(* LS Electric XG5000 project: 11_01_project *)
(* PLC LSPLC *)

PROGRAM NewProgram (* task: 스캔 프로그램 *)
VAR
    dd : BOOL;
    ET : TIME;
    INST : TON;
    INST1 : TP;
    INST10 : TON;
    INST11 : TMR_FLK;
    INST12 : TON;
    INST13 : TMR_FLK;
    INST14 : TOF;
    INST15 : TOF;
    INST16 : TOF;
    INST17 : TOF;
    INST18 : CTD_INT;
    INST19 : CTD_INT;
    INST2 : TP;
    INST20 : TMR_FLK;
    INST21 : TMR_FLK;
    INST22 : TOF;
    INST23 : CTD_INT;
    INST3 : TON;
    INST4 : TP;
    INST5 : TP_RST;
    INST6 : TP;
    INST7 : TMR_FLK;
    INST8 : TP;
    INST9 : TMR_FLK;
    intcv : BOOL;
    LD : BOOL;
    RST : BOOL;
    ㄱㄱ : BOOL;
    걍 : BOOL;
END_VAR

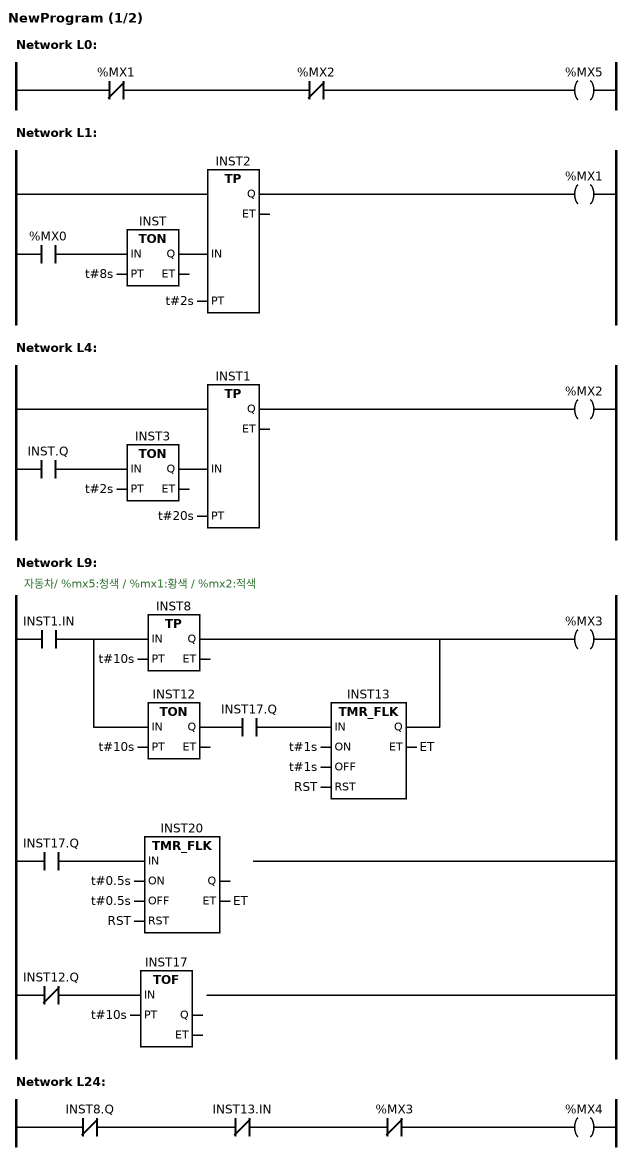
(* Rung L0 *)
%MX5 := NOT %MX1 AND NOT %MX2;
(* Rung L1 *)
INST(IN := %MX0, PT := t#8s);
INST2(IN := INST.Q, PT := t#2s);
%MX1 := INST2.Q;
(* Rung L4 *)
INST3(IN := INST.Q, PT := t#2s);
INST1(IN := INST3.Q, PT := t#20s);
%MX2 := INST1.Q;
(* 자동차/ %mx5:청색 / %mx1:황색 / %mx2:적색 *)
(* Rung L9 *)
INST8(IN := INST1.IN, PT := t#10s);
INST12(IN := INST1.IN, PT := t#10s);
INST13(IN := INST12.Q AND INST17.Q, ON := t#1s, OFF := t#1s, RST := RST, ET => ET);
%MX3 := INST8.Q OR INST13.Q;
INST20(IN := INST17.Q, ON := t#0.5s, OFF := t#0.5s, RST := RST, ET => ET);
INST17(IN := NOT INST12.Q, PT := t#10s);
(* Rung L24 *)
%MX4 := NOT INST8.Q AND NOT INST13.IN AND NOT %MX3;

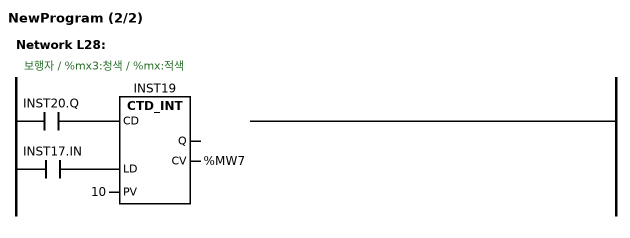
(* 보행자 / %mx3:청색 / %mx:적색 *)
(* Rung L28 *)
INST19(CD := INST20.Q, LD := INST17.IN, PV := 10, CV => %MW7);
(* 카운터 *)
END_PROGRAM